INTERFACE I_Axis_BaseUnit EXTENDS I_ResourceLock

PROPERTY AxisActualPosition : LREAL
GET
END_GET
END_PROPERTY

PROPERTY AxisActualVelocity : LREAL
GET
END_GET
END_PROPERTY

PROPERTY AxisHasJob : BOOL
GET
END_GET
END_PROPERTY

PROPERTY AxisIsDisabled : BOOL
GET
END_GET
END_PROPERTY

METHOD M_CyclicUpdate
VAR_INPUT
END_VAR
END_METHOD

METHOD M_Halt : BOOL
VAR_INPUT
	OwnerId : T_ResourceOwnerId;
	Execute : BOOL;
	Deceleration : LREAL;
END_VAR
VAR_OUTPUT
	Done : BOOL;
	Error : BOOL;
END_VAR
END_METHOD

METHOD M_Jog : BOOL
VAR_INPUT
	OwnerId : T_ResourceOwnerId;
	JogForward : BOOL;
	JogBackwards : BOOL;
	Mode : E_JogMode;
	Position : LREAL;
	Velocity : LREAL;
	Acceleration : LREAL;
	Deceleration : LREAL;
END_VAR
VAR_OUTPUT
	Done : BOOL;
	Error : BOOL;
	ErrorId : UDINT;
END_VAR
END_METHOD

METHOD M_MoveAbs : BOOL
VAR_INPUT
	OwnerId : T_ResourceOwnerId;
	Execute : BOOL;
	Position : LREAL;
	Velocity : LREAL;
	Acceleration : LREAL;
	Deceleration : LREAL;
END_VAR
VAR_OUTPUT
	Done : BOOL;
	Error : BOOL;
	ErrorId : UDINT;
END_VAR
END_METHOD

METHOD M_MoveVel : BOOL
VAR_INPUT
	OwnerId : T_ResourceOwnerId;
	Execute : BOOL;
	Direction : MC_Direction;
	Velocity : LREAL;
	Acceleration : LREAL;
	Deceleration : LREAL;
END_VAR
VAR_OUTPUT
	InVelocity : BOOL;
	Error : BOOL;
END_VAR
END_METHOD

METHOD M_Reset : BOOL
VAR_INPUT
	OwnerId : T_ResourceOwnerId;
	Execute : BOOL;
END_VAR
VAR_OUTPUT
	Done : BOOL;
	Error : BOOL;
	ErrorId : UDINT;
END_VAR
END_METHOD

METHOD M_Stop : BOOL
VAR_INPUT
	OwnerId : T_ResourceOwnerId;
	Execute : BOOL;
	Deceleration : LREAL;
END_VAR
VAR_OUTPUT
	Done : BOOL;
	Error : BOOL;
	ErrorId : UDINT;
END_VAR
END_METHOD

END_INTERFACE

(* stored: Version 1.1.0.1, ProductVersion 3.1.4026.18
   Itf I_Axis_BaseUnit: Id {6467168b-19d5-4331-8d22-d28396010198}
   Property AxisActualPosition: Id {eab3f334-68f5-41a8-941d-f2167723f8cf}
   Get Get: Id {c87b0730-c36b-45e0-ad8a-c20fe11aeef8}
   Property AxisActualVelocity: Id {21e250a2-5522-44f8-b388-4567d023dbfe}
   Get Get: Id {84b28254-08aa-419a-a385-ea8b63e47b57}
   Property AxisHasJob: Id {a1938803-7419-476d-8402-590d311440cf}
   Get Get: Id {f06a2727-a7b5-40e3-8e1f-b665de9846da}
   Property AxisIsDisabled: Id {2d6192b0-67ac-40f2-b5fa-6a71916a4e40}
   Get Get: Id {08c167f8-c5d6-4bf5-ae04-4d1f31fbeb0c}
   Method M_CyclicUpdate: Id {1cba92c4-21e1-4f38-a0a3-633174eef5ec}
   Method M_Halt: Id {1794374f-bb34-4f57-8d42-269a47ec9875}
   Method M_Jog: Id {8ddc2b2f-0491-430c-bacb-ff55df4dc1d4}
   Method M_MoveAbs: Id {f9a6b842-1791-47c1-8b12-947d9ce6b1ac}
   Method M_MoveVel: Id {3866eee3-20c5-488f-bb14-447afbad6b44}
   Method M_Reset: Id {8fe19313-b7c2-4cbf-a8f1-cb5cb030e7af}
   Method M_Stop: Id {b848d1e0-db43-4d37-93f3-46b8e8154c0b} *)
